// TIA Portal V20 export
PlcWatchTable "Fx_OnlineWatch"
  PlcWatchTableEntry   Address=%M0.0, DisplayFormat=Bool, Comment="Fixture row 1"
  PlcWatchTableEntry   Address=%MW2, DisplayFormat=Hex, Comment="Fixture row 2"
  PlcWatchTableEntry   Address=%ID0, DisplayFormat=Hex, Comment="Fixture row 3"
  PlcWatchTableEntry   Address=%QB4, DisplayFormat=Hex, Comment="Fixture row 4"
  PlcWatchTableEntry ""Fx_Global".Count"  DisplayFormat=DEC_signed, ModifyValue=17, Comment="Fixture row 5"
  PlcWatchTableEntry ""Fx_Global".Ready"  DisplayFormat=Bool, Comment="Fixture row 6"
  PlcWatchTableEntry ""Fx_Global".Count"  DisplayFormat=DEC_signed, Comment="Fixture row 7"
